FUNCTION "ST10Cyl_interface91-100" : Void
VAR_INPUT
  AlwaysON : Bool;
  E_stop : Bool;
END_VAR
VAR_TEMP
  tTest : Bool;
END_VAR
BEGIN
  // Původní jazyk: LAD
  // Zdroj XML: EXPORT/Program blocks/OP010/10_Device/01_Cylinder/ST10Cyl_interface91-100.xml
  // --- LAD/FBD → SCL (orientační převod, jen pro revizi) ---
  // Network 1
  ST10Cylinder.Cy := (#AlwaysON AND #E_stop);
  ST10Cylinder.Cy := (#AlwaysON AND #E_stop);
  ST10Cylinder.Cy := (#AlwaysON AND NOT #AlwaysON);
  // Network 2
  ST10Cylinder.Cy := (#AlwaysON AND #E_stop);
  ST10Cylinder.Cy := (#AlwaysON AND #E_stop);
  ST10Cylinder.Cy := (#AlwaysON AND NOT #AlwaysON);
  // Network 3
  ST10Cylinder.Cy := (#AlwaysON AND #E_stop);
  ST10Cylinder.Cy := (#AlwaysON AND #E_stop);
  ST10Cylinder.Cy := (#AlwaysON AND NOT #AlwaysON);
  // Network 4
  ST10Cylinder.Cy := (#AlwaysON AND #E_stop);
  ST10Cylinder.Cy := (#AlwaysON AND #E_stop);
  ST10Cylinder.Cy := (#AlwaysON AND NOT #AlwaysON);
  // Network 5
  ST10Cylinder.Cy := (#AlwaysON AND #E_stop);
  ST10Cylinder.Cy := (#AlwaysON AND #E_stop);
  ST10Cylinder.Cy := (#AlwaysON AND NOT #AlwaysON);
  // Network 6
  ST10Cylinder.Cy := (#AlwaysON AND #E_stop);
  ST10Cylinder.Cy := (#AlwaysON AND #E_stop);
  ST10Cylinder.Cy := (#AlwaysON AND NOT #AlwaysON);
  // Network 7
  ST10Cylinder.Cy := (#AlwaysON AND #E_stop);
  ST10Cylinder.Cy := (#AlwaysON AND #E_stop);
  ST10Cylinder.Cy := (#AlwaysON AND NOT #AlwaysON);
  // Network 8
  ST10Cylinder.Cy := (#AlwaysON AND #E_stop);
  ST10Cylinder.Cy := (#AlwaysON AND #E_stop);
  ST10Cylinder.Cy := (#AlwaysON AND NOT #AlwaysON);
  // Network 9
  ST10Cylinder.Cy := (#AlwaysON AND #E_stop);
  ST10Cylinder.Cy := (#AlwaysON AND #E_stop);
  ST10Cylinder.Cy := (#AlwaysON AND NOT #AlwaysON);
  // Network 10
  ST10Cylinder.Cy := (#AlwaysON AND #E_stop);
  ST10Cylinder.Cy := (#AlwaysON AND #E_stop);
  ST10Cylinder.Cy := (#AlwaysON AND NOT #AlwaysON);
END_FUNCTION
